{attribute 'linkalways'}
{attribute 'no_explicit_call' := 'This FB is a CLASS and must be accessed using methods or properties'}
{attribute 'enable_dynamic_creation'}
FUNCTION_BLOCK _TcVnParamsWalshBarcodeDetection EXTENDS StructuredDatatypeBase
VAR
    localData : TcVnParamsWalshBarcodeDetection := (nMaxBarDistance := 8, fMinAspectRatio := 1.0, fMaxAspectRatio := 5.0, nIntensityDifference := 100, nMinArea := -1, nChannelIndex := -1, nWalshFilterNum := 5, fOutlierReductionFactor := 1.0, fBarConnectionFactor := 1.0, fRegionFilterFactor := 1.0, fPostProcessingResizeFactor := 0.5, eInterpolationType := TCVN_IT_BILINEAR);
    activeData : REFERENCE TO TcVnParamsWalshBarcodeDetection REF= localData;
    _nMaxBarDistance : _UDINT(localData.nMaxBarDistance);
    _fMinAspectRatio : _REAL(localData.fMinAspectRatio);
    _fMaxAspectRatio : _REAL(localData.fMaxAspectRatio);
    _nIntensityDifference : _UDINT(localData.nIntensityDifference);
    _nMinArea : _DINT(localData.nMinArea);
    _nChannelIndex : _DINT(localData.nChannelIndex);
    _nWalshFilterNum : _UDINT(localData.nWalshFilterNum);
    _fOutlierReductionFactor : _REAL(localData.fOutlierReductionFactor);
    _fBarConnectionFactor : _REAL(localData.fBarConnectionFactor);
    _fRegionFilterFactor : _REAL(localData.fRegionFilterFactor);
    _fPostProcessingResizeFactor : _REAL(localData.fPostProcessingResizeFactor);
    _eInterpolationType : _ETcVnInterpolationType(localData.eInterpolationType);
END_VAR

PROPERTY PUBLIC Address : PVOID
GET
Address := ADR(activeData);
END_GET
END_PROPERTY

METHOD PUBLIC ClearReference
VAR_INPUT
END_VAR
activeData REF= localData;
SetMemberReference();
END_METHOD

METHOD PUBLIC Clone : I_Datatype
VAR
    pClone : POINTER TO _TcVnParamsWalshBarcodeDetection;
END_VAR
pClone := __NEW(_TcVnParamsWalshBarcodeDetection);
IF pClone = 0 THEN
    RETURN;
END_IF
pClone^.TryCopyFrom(THIS^);
Clone := pClone^;
END_METHOD

METHOD FB_init : BOOL
VAR_INPUT
	bInitRetains : BOOL; // if TRUE, the retain variables are initialized (warm start / cold start)
	bInCopyCode : BOOL;  // if TRUE, the instance afterwards gets moved into the copy code (online change)
END_VAR
SetMemberReference();
AddMember('nMaxBarDistance', _nMaxBarDistance);
AddMember('fMinAspectRatio', _fMinAspectRatio);
AddMember('fMaxAspectRatio', _fMaxAspectRatio);
AddMember('nIntensityDifference', _nIntensityDifference);
AddMember('nMinArea', _nMinArea);
AddMember('nChannelIndex', _nChannelIndex);
AddMember('nWalshFilterNum', _nWalshFilterNum);
AddMember('fOutlierReductionFactor', _fOutlierReductionFactor);
AddMember('fBarConnectionFactor', _fBarConnectionFactor);
AddMember('fRegionFilterFactor', _fRegionFilterFactor);
AddMember('fPostProcessingResizeFactor', _fPostProcessingResizeFactor);
AddMember('eInterpolationType', _eInterpolationType);
END_METHOD

PROPERTY PUBLIC Identifier : T_MAXSTRING
GET
Identifier := 'TcVnParamsWalshBarcodeDetection';
END_GET
END_PROPERTY

METHOD PUBLIC MakeReferenceTo
VAR_INPUT
	ReferenceTarget : REFERENCE TO TcVnParamsWalshBarcodeDetection;
END_VAR
activeData REF= ReferenceTarget;
SetMemberReference();
END_METHOD

METHOD PROTECTED SetMemberReference
VAR_INPUT
END_VAR
_nMaxBarDistance.MakeReferenceTo(activeData.nMaxBarDistance);
_fMinAspectRatio.MakeReferenceTo(activeData.fMinAspectRatio);
_fMaxAspectRatio.MakeReferenceTo(activeData.fMaxAspectRatio);
_nIntensityDifference.MakeReferenceTo(activeData.nIntensityDifference);
_nMinArea.MakeReferenceTo(activeData.nMinArea);
_nChannelIndex.MakeReferenceTo(activeData.nChannelIndex);
_nWalshFilterNum.MakeReferenceTo(activeData.nWalshFilterNum);
_fOutlierReductionFactor.MakeReferenceTo(activeData.fOutlierReductionFactor);
_fBarConnectionFactor.MakeReferenceTo(activeData.fBarConnectionFactor);
_fRegionFilterFactor.MakeReferenceTo(activeData.fRegionFilterFactor);
_fPostProcessingResizeFactor.MakeReferenceTo(activeData.fPostProcessingResizeFactor);
_eInterpolationType.MakeReferenceTo(activeData.eInterpolationType);
END_METHOD

PROPERTY PUBLIC Size : UDINT
GET
Size := SIZEOF(activeData);
END_GET
END_PROPERTY

METHOD TryMakeReferenceTo : BOOL
VAR_INPUT
	Target : I_Datatype;
END_VAR
VAR
	pTargetData : POINTER TO TcVnParamsWalshBarcodeDetection;
END_VAR
IF NOT IsEquivalentTo(Target) THEN
	RETURN;
END_IF

pTargetData := Target.Address;
activeData REF= pTargetData^;
SetMemberReference();
TryMakeReferenceTo := TRUE;
END_METHOD

PROPERTY PUBLIC Value : REFERENCE TO TcVnParamsWalshBarcodeDetection
GET
Value REF= activeData;
END_GET
END_PROPERTY

PROPERTY PUBLIC nMaxBarDistance : REFERENCE TO _UDINT
GET
nMaxBarDistance REF= _nMaxBarDistance;
END_GET
END_PROPERTY

PROPERTY PUBLIC fMinAspectRatio : REFERENCE TO _REAL
GET
fMinAspectRatio REF= _fMinAspectRatio;
END_GET
END_PROPERTY

PROPERTY PUBLIC fMaxAspectRatio : REFERENCE TO _REAL
GET
fMaxAspectRatio REF= _fMaxAspectRatio;
END_GET
END_PROPERTY

PROPERTY PUBLIC nIntensityDifference : REFERENCE TO _UDINT
GET
nIntensityDifference REF= _nIntensityDifference;
END_GET
END_PROPERTY

PROPERTY PUBLIC nMinArea : REFERENCE TO _DINT
GET
nMinArea REF= _nMinArea;
END_GET
END_PROPERTY

PROPERTY PUBLIC nChannelIndex : REFERENCE TO _DINT
GET
nChannelIndex REF= _nChannelIndex;
END_GET
END_PROPERTY

PROPERTY PUBLIC nWalshFilterNum : REFERENCE TO _UDINT
GET
nWalshFilterNum REF= _nWalshFilterNum;
END_GET
END_PROPERTY

PROPERTY PUBLIC fOutlierReductionFactor : REFERENCE TO _REAL
GET
fOutlierReductionFactor REF= _fOutlierReductionFactor;
END_GET
END_PROPERTY

PROPERTY PUBLIC fBarConnectionFactor : REFERENCE TO _REAL
GET
fBarConnectionFactor REF= _fBarConnectionFactor;
END_GET
END_PROPERTY

PROPERTY PUBLIC fRegionFilterFactor : REFERENCE TO _REAL
GET
fRegionFilterFactor REF= _fRegionFilterFactor;
END_GET
END_PROPERTY

PROPERTY PUBLIC fPostProcessingResizeFactor : REFERENCE TO _REAL
GET
fPostProcessingResizeFactor REF= _fPostProcessingResizeFactor;
END_GET
END_PROPERTY

PROPERTY PUBLIC eInterpolationType : REFERENCE TO _ETcVnInterpolationType
GET
eInterpolationType REF= _eInterpolationType;
END_GET
END_PROPERTY

END_FUNCTION_BLOCK

(* stored: Version 1.1.0.1, ProductVersion 3.1.4024.13
   POU _TcVnParamsWalshBarcodeDetection: Id {fe845983-f29f-4b44-8ff0-01de82ebe09a}, SpecialFunc None
   Folder Core: Id {57b274cb-9684-41b4-ab65-0d0202f7b4e9}
   Folder Customize: Id {9beafbe5-9c27-4395-9731-d6a0513786bc}
   Folder Constructor: Id {e6f11ef6-cfaa-4661-974b-468f4b35313e}
   Folder Protected: Id {c94b7c7e-d391-47b3-b63e-0ad65fe9173a}
   Property Address: Id {16103200-3a49-4a5e-952b-3cfc14118e2b}
   Get Get: Id {936d103b-2d1f-4b74-ac48-298bd103fb83}
   Method ClearReference: Id {2cf9d87b-978f-4701-9cf1-dbafd005b847}
   Method Clone: Id {623ed220-dbe2-413b-b3a4-5add0d2ee25e}
   Method FB_init: Id {1cdbfddd-cac4-4945-912c-39ab76f2b176}
   Property Identifier: Id {f4cd0b96-cade-483a-88d6-a13cecb65635}
   Get Get: Id {47e84d38-581b-42fe-84f5-c31547f28eb5}
   Method MakeReferenceTo: Id {3539b1df-ba34-483a-8e36-b26784182cba}
   Method SetMemberReference: Id {d8c6e286-a035-4864-b7cd-f81489d86489}
   Property Size: Id {00bb9efc-5bc3-4061-bd9f-86312d86b1a3}
   Get Get: Id {c76adae4-8839-4d32-a79d-5dfb2e63542f}
   Method TryMakeReferenceTo: Id {9ac639f8-b4d9-47a1-91a3-eb88273b99b8}
   Property Value: Id {b7412016-aa78-49ea-858b-8fce6b6080b1}
   Get Get: Id {75cd579d-313b-4436-9d77-4ca439f82f0e}
   Property nMaxBarDistance: Id {950a35ca-f4dd-4398-9cb4-0a3d636daec4}
   Get Get: Id {fc8129df-0f77-4f81-acc2-4b4b29caafaa}
   Property fMinAspectRatio: Id {94795c55-06a6-46ec-bf11-82347bd13a9f}
   Get Get: Id {546e8059-2296-4159-a553-e12452f0c6f5}
   Property fMaxAspectRatio: Id {248a4bc2-4a5a-4df1-8f14-f21100454d24}
   Get Get: Id {684668ea-bb06-461a-8491-0029dec00d4b}
   Property nIntensityDifference: Id {fcd96c14-bcb6-4bb8-8f5b-00b4c3f5b706}
   Get Get: Id {12ed7c96-1d9f-4629-9d2b-ad04d0394449}
   Property nMinArea: Id {28814f8a-5838-41e4-9af0-8fd9d98d2b3e}
   Get Get: Id {40d119da-9518-421b-8577-6162785defe6}
   Property nChannelIndex: Id {2d2f75fd-7525-40c4-99cb-aeb450fcd982}
   Get Get: Id {4abfb8f6-f6bc-4bc6-8aea-661d36bebb23}
   Property nWalshFilterNum: Id {08ca4838-dd81-4bb0-8f38-5133924d6809}
   Get Get: Id {57c8cec2-ec38-46e6-8c93-8915b7cbde6f}
   Property fOutlierReductionFactor: Id {44985f94-47ef-4bc2-a4a9-8741cad74753}
   Get Get: Id {24d725ca-4ea4-4b97-8710-a6023b3e55e0}
   Property fBarConnectionFactor: Id {21089076-d624-4a51-a013-95edc755ab97}
   Get Get: Id {1947d76e-08ed-4b88-86ed-d12d3fbac69b}
   Property fRegionFilterFactor: Id {7d72bebf-f436-4b48-adb6-003988925fae}
   Get Get: Id {59771fee-b5fe-45e2-adf8-b7de7730b7a7}
   Property fPostProcessingResizeFactor: Id {f56a8d53-b94d-4b44-8adb-e5ccaf0c74fb}
   Get Get: Id {1483168a-15b8-4a87-89cc-883c7a62e374}
   Property eInterpolationType: Id {84799021-67cd-489c-95a6-8a96b2a8688c}
   Get Get: Id {5ba4265f-6f7c-4bd1-b8c1-696bb4cdd458} *)
